(* LS Electric XG5000 project: Three_Guys_Plc *)
(* PLC LSPLC *)
(* module base 0 slot 0: FEnet:XGL-EFMT(B) (Fast Ethernet 통신 모듈, 전기 Master) *)
(* module base 0 slot 1: 입력 모듈:XGI-A21A/C (AC 220V 입력, 8점(8점/COM) / 8점(1점/COM)) *)
(* module base 0 slot 2: 출력 모듈:XGQ-RY1A (릴레이 출력, 8점 (2A용, 단독 COM.)) *)

PROGRAM HeatTreatPlc (* task: 스캔 프로그램 *)
VAR
    ENO : BOOL;
    곱하기60 : TIME := T#60s;
    기계1_가스_밸브 AT %MX8010 : BOOL;
    기계1_가스이상램프 AT %MX8011 : BOOL;
    기계1_가스이상센서 AT %MX8061 : BOOL;
    기계1_가열_min : TIME;
    기계1_가열_시간 AT %MD506 : DWORD;
    기계1_가열냉각_시간 : TIME;
    기계1_가열시간설정 : TOF;
    기계1_경고 AT %MX8019 : BOOL;
    기계1_경과시간_msec : TIME;
    기계1_남은시간_min AT %MD509 : TIME;
    기계1_남은시간_msec : TIME;
    기계1_냉각_min : TIME;
    기계1_냉각_밸브 AT %MX8012 : BOOL;
    기계1_냉각_시간 AT %MD507 : DWORD;
    기계1_냉각시간설정 : TOF;
    기계1_냉각이상램프 AT %MX8013 : BOOL;
    기계1_냉각이상센서 AT %MX8062 : BOOL;
    기계1_문 AT %MX8016 : BOOL;
    기계1_문ON_타이머 : TON;
    기계1_문이상램프 AT %MX8017 : BOOL;
    기계1_문이상센서 AT %MX8064 : BOOL;
    기계1_설정온도입력 AT %MW1010 : WORD;
    기계1_열선 AT %MX8014 : BOOL;
    기계1_열선이상램프 AT %MX8015 : BOOL;
    기계1_열선이상센서 AT %MX8063 : BOOL;
    기계1_작동 AT %MX8018 : BOOL;
    기계1_전원 AT %MX8001 : BOOL;
    기계1_중지 AT %MX8020 : BOOL;
    기계1_현재질화로온도 AT %MW1016 : WORD := 100;
    기계2_가스_밸브 AT %MX9010 : BOOL;
    기계2_가스이상램프 AT %MX9011 : BOOL;
    기계2_가스이상센서 AT %MX9061 : BOOL;
    기계2_가열_min : TIME;
    기계2_가열_시간 AT %MD569 : DWORD;
    기계2_가열냉각_시간 : TIME;
    기계2_가열시간설정 : TOF;
    기계2_경고 AT %MX9019 : BOOL;
    기계2_경과시간_msec : TIME;
    기계2_남은시간_min AT %MD572 : TIME;
    기계2_남은시간_msec : TIME;
    기계2_냉각_min : TIME;
    기계2_냉각_밸브 AT %MX9012 : BOOL;
    기계2_냉각_시간 AT %MD570 : DWORD;
    기계2_냉각시간설정 : TOF;
    기계2_냉각이상램프 AT %MX9013 : BOOL;
    기계2_냉각이상센서 AT %MX9062 : BOOL;
    기계2_문 AT %MX9016 : BOOL;
    기계2_문ON_타이머 : TON;
    기계2_문이상램프 AT %MX9017 : BOOL;
    기계2_문이상센서 AT %MX9064 : BOOL;
    기계2_설정온도입력 AT %MW1136 : WORD;
    기계2_열선 AT %MX9014 : BOOL;
    기계2_열선이상램프 AT %MX9015 : BOOL;
    기계2_열선이상센서 AT %MX9063 : BOOL;
    기계2_작동 AT %MX9018 : BOOL;
    기계2_전원 AT %MX9001 : BOOL;
    기계2_중지 AT %MX9020 : BOOL;
    기계2_현재질화로온도 AT %MW1142 : WORD;
    기계3_가스_밸브 AT %MX10010 : BOOL;
    기계3_가스이상램프 AT %MX10011 : BOOL;
    기계3_가스이상센서 AT %MX10061 : BOOL;
    기계3_가열_min : TIME;
    기계3_가열_시간 AT %MD631 : DWORD;
    기계3_가열냉각_시간 : TIME;
    기계3_가열시간설정 : TOF;
    기계3_경고 AT %MX10019 : BOOL;
    기계3_경과시간_msec : TIME;
    기계3_남은시간_min AT %MD634 : TIME;
    기계3_남은시간_msec : TIME;
    기계3_냉각_min : TIME;
    기계3_냉각_밸브 AT %MX10012 : BOOL;
    기계3_냉각_시간 AT %MD632 : DWORD;
    기계3_냉각시간설정 : TOF;
    기계3_냉각이상램프 AT %MX10013 : BOOL;
    기계3_냉각이상센서 AT %MX10062 : BOOL;
    기계3_문 AT %MX10016 : BOOL;
    기계3_문ON_타이머 : TON;
    기계3_문이상램프 AT %MX10017 : BOOL;
    기계3_문이상센서 AT %MX10064 : BOOL;
    기계3_설정온도입력 AT %MW1260 : WORD;
    기계3_열선 AT %MX10014 : BOOL;
    기계3_열선이상램프 AT %MX10015 : BOOL;
    기계3_열선이상센서 AT %MX10063 : BOOL;
    기계3_작동 AT %MX10018 : BOOL;
    기계3_전원 AT %MX10001 : BOOL;
    기계3_중지 AT %MX10020 : BOOL;
    기계3_현재질화로온도 AT %MW1266 : WORD;
    기계4_가스_밸브 AT %MX11010 : BOOL;
    기계4_가스이상램프 AT %MX11011 : BOOL;
    기계4_가스이상센서 AT %MX11061 : BOOL;
    기계4_가열_min : TIME;
    기계4_가열_시간 AT %MD694 : DWORD;
    기계4_가열냉각_시간 : TIME;
    기계4_가열시간설정 : TOF;
    기계4_경고 AT %MX11019 : BOOL;
    기계4_경과시간_msec : TIME;
    기계4_남은시간_min AT %MD697 : TIME;
    기계4_남은시간_msec : TIME;
    기계4_냉각_min : TIME;
    기계4_냉각_밸브 AT %MX11012 : BOOL;
    기계4_냉각_시간 AT %MD695 : DWORD;
    기계4_냉각시간설정 : TOF;
    기계4_냉각이상램프 AT %MX11013 : BOOL;
    기계4_냉각이상센서 AT %MX11062 : BOOL;
    기계4_문 AT %MX11016 : BOOL;
    기계4_문ON_타이머 : TON;
    기계4_문이상램프 AT %MX11017 : BOOL;
    기계4_문이상센서 AT %MX11064 : BOOL;
    기계4_설정온도입력 AT %MW1386 : WORD;
    기계4_열선 AT %MX11014 : BOOL;
    기계4_열선이상램프 AT %MX11015 : BOOL;
    기계4_열선이상센서 AT %MX11063 : BOOL;
    기계4_작동 AT %MX11018 : BOOL;
    기계4_전원 AT %MX11001 : BOOL;
    기계4_중지 AT %MX11020 : BOOL;
    기계4_현재질화로온도 AT %MW1392 : WORD;
    기계_신호기 : TP;
    기계_신호기1 : TP;
    기계_신호기2 : TP;
    기계_신호기3 : TP;
END_VAR
VAR
    _p1 : BOOL;
    _e2 : R_TRIG;
    _e3 : F_TRIG;
    _p4 : BOOL;
    _e5 : R_TRIG;
    _e6 : F_TRIG;
    _p7 : BOOL;
    _e8 : R_TRIG;
    _e9 : F_TRIG;
    _p10 : BOOL;
    _e11 : R_TRIG;
    _e12 : F_TRIG;
    _p13 : BOOL;
    _e14 : R_TRIG;
    _t15 : BOOL;
    _e16 : R_TRIG;
    _p17 : BOOL;
    _e18 : R_TRIG;
    _e19 : F_TRIG;
    _p20 : BOOL;
    _e21 : R_TRIG;
    _e22 : F_TRIG;
    _p23 : BOOL;
    _e24 : R_TRIG;
    _e25 : F_TRIG;
    _p26 : BOOL;
    _e27 : R_TRIG;
    _e28 : F_TRIG;
    _p29 : BOOL;
    _e30 : R_TRIG;
    _t31 : BOOL;
    _e32 : R_TRIG;
    _p33 : BOOL;
    _e34 : R_TRIG;
    _e35 : F_TRIG;
    _p36 : BOOL;
    _e37 : R_TRIG;
    _e38 : F_TRIG;
    _p39 : BOOL;
    _e40 : R_TRIG;
    _e41 : F_TRIG;
    _p42 : BOOL;
    _e43 : R_TRIG;
    _e44 : F_TRIG;
    _p45 : BOOL;
    _e46 : R_TRIG;
    _t47 : BOOL;
    _e48 : R_TRIG;
    _p49 : BOOL;
    _e50 : R_TRIG;
    _e51 : F_TRIG;
    _p52 : BOOL;
    _e53 : R_TRIG;
    _e54 : F_TRIG;
    _p55 : BOOL;
    _e56 : R_TRIG;
    _e57 : F_TRIG;
    _p58 : BOOL;
    _e59 : R_TRIG;
    _e60 : F_TRIG;
    _p61 : BOOL;
    _e62 : R_TRIG;
    _t63 : BOOL;
    _e64 : R_TRIG;
END_VAR

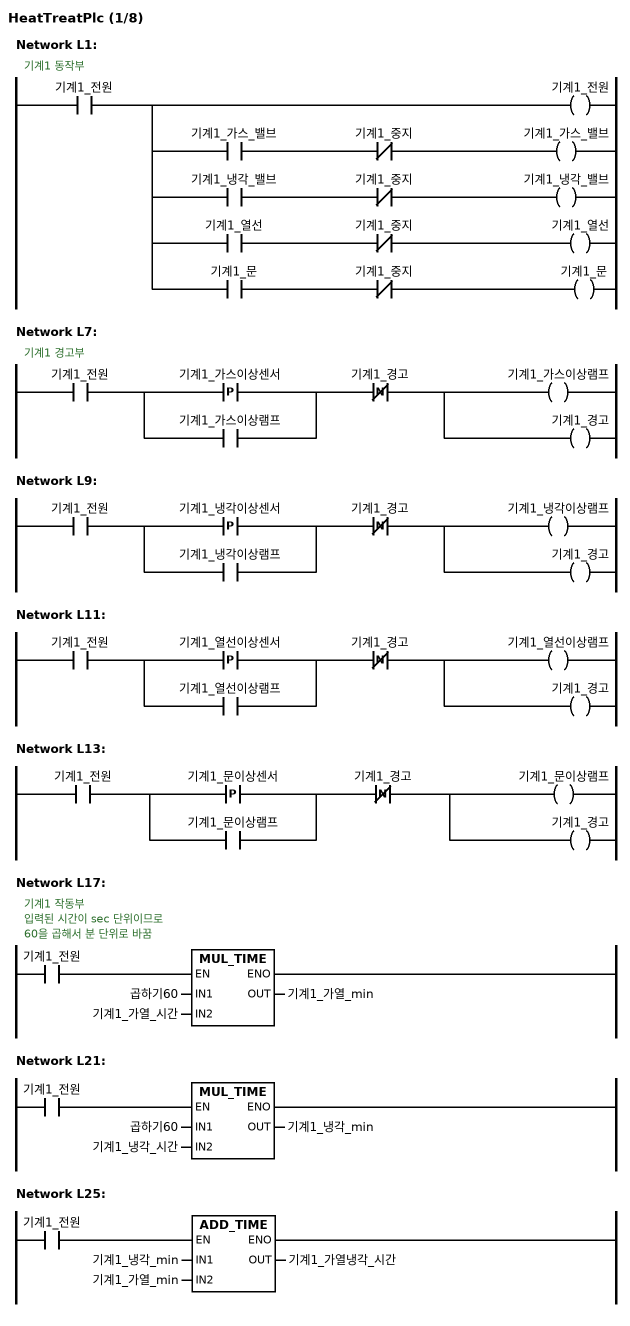
(* 기계1 동작부 *)
(* Rung L1 *)
_p1 := 기계1_전원;
기계1_전원 := _p1;
기계1_가스_밸브 := _p1 AND 기계1_가스_밸브 AND NOT 기계1_중지;
기계1_냉각_밸브 := _p1 AND 기계1_냉각_밸브 AND NOT 기계1_중지;
기계1_열선 := _p1 AND 기계1_열선 AND NOT 기계1_중지;
기계1_문 := _p1 AND 기계1_문 AND NOT 기계1_중지;
(* 기계1 경고부 *)
(* Rung L7 *)
_e2(CLK := 기계1_가스이상센서);
_e3(CLK := 기계1_경고);
_p4 := 기계1_전원 AND (_e2.Q OR 기계1_가스이상램프) AND NOT _e3.Q;
기계1_가스이상램프 := _p4;
기계1_경고 := _p4;
(* Rung L9 *)
_e5(CLK := 기계1_냉각이상센서);
_e6(CLK := 기계1_경고);
_p7 := 기계1_전원 AND (_e5.Q OR 기계1_냉각이상램프) AND NOT _e6.Q;
기계1_냉각이상램프 := _p7;
기계1_경고 := _p7;
(* Rung L11 *)
_e8(CLK := 기계1_열선이상센서);
_e9(CLK := 기계1_경고);
_p10 := 기계1_전원 AND (_e8.Q OR 기계1_열선이상램프) AND NOT _e9.Q;
기계1_열선이상램프 := _p10;
기계1_경고 := _p10;
(* Rung L13 *)
_e11(CLK := 기계1_문이상센서);
_e12(CLK := 기계1_경고);
_p13 := 기계1_전원 AND (_e11.Q OR 기계1_문이상램프) AND NOT _e12.Q;
기계1_문이상램프 := _p13;
기계1_경고 := _p13;
(* 기계1 작동부 *)
(* 입력된 시간이 sec 단위이므로 / 60을 곱해서 분 단위로 바꿈 *)
(* Rung L17 *)
IF 기계1_전원 THEN 기계1_가열_min := MUL_TIME(곱하기60, 기계1_가열_시간); END_IF;
(* Rung L21 *)
IF 기계1_전원 THEN 기계1_냉각_min := MUL_TIME(곱하기60, 기계1_냉각_시간); END_IF;
(* Rung L25 *)
IF 기계1_전원 THEN 기계1_가열냉각_시간 := ADD_TIME(기계1_냉각_min, 기계1_가열_min); END_IF;

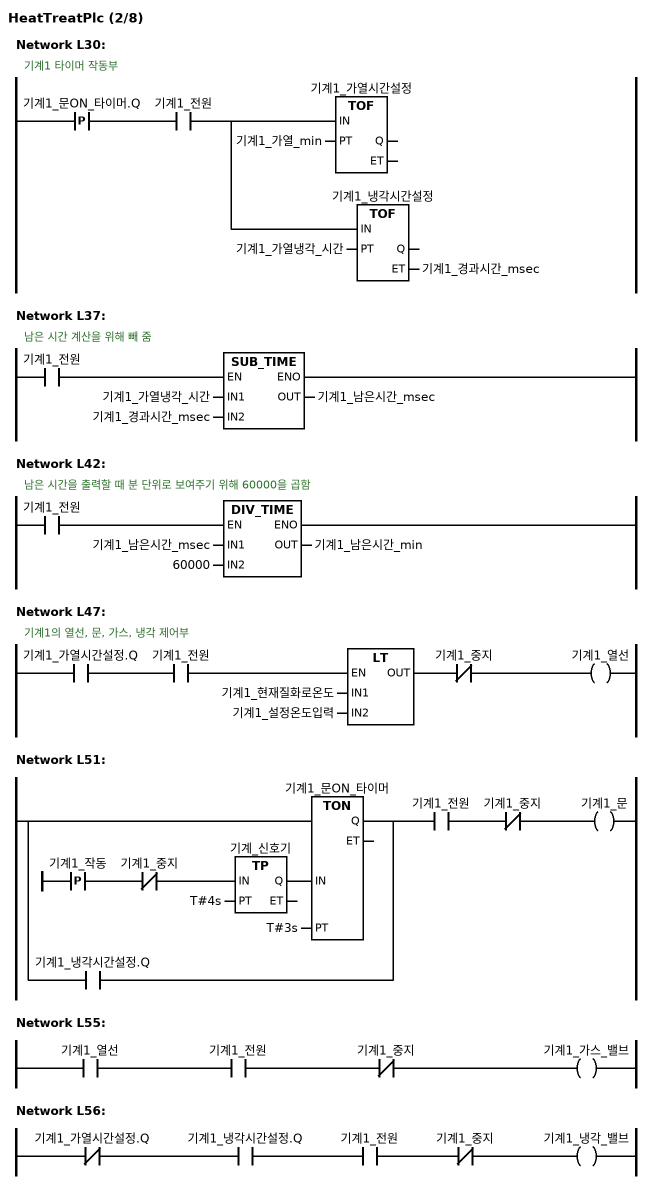
(* 기계1 타이머 작동부 *)
(* Rung L30 *)
_e14(CLK := 기계1_문ON_타이머.Q);
기계1_가열시간설정(IN := _e14.Q AND 기계1_전원, PT := 기계1_가열_min);
기계1_냉각시간설정(IN := _e14.Q AND 기계1_전원, PT := 기계1_가열냉각_시간, ET => 기계1_경과시간_msec);
(* 남은 시간 계산을 위해 빼 줌 *)
(* Rung L37 *)
IF 기계1_전원 THEN 기계1_남은시간_msec := SUB_TIME(기계1_가열냉각_시간, 기계1_경과시간_msec); END_IF;
(* 남은 시간을 출력할 때 분 단위로 보여주기 위해 60000을 곱함 *)
(* Rung L42 *)
IF 기계1_전원 THEN 기계1_남은시간_min := DIV_TIME(기계1_남은시간_msec, 60000); END_IF;
(* 기계1의 열선, 문, 가스, 냉각 제어부 *)
(* Rung L47 *)
IF 기계1_가열시간설정.Q AND 기계1_전원 THEN _t15 := 기계1_현재질화로온도 < 기계1_설정온도입력; END_IF;
기계1_열선 := _t15 AND NOT 기계1_중지;
(* Rung L51 *)
_e16(CLK := 기계1_작동);
기계_신호기(IN := _e16.Q AND NOT 기계1_중지, PT := T#4s);
기계1_문ON_타이머(IN := 기계_신호기.Q, PT := T#3s);
기계1_문 := (기계1_문ON_타이머.Q OR 기계1_냉각시간설정.Q) AND 기계1_전원 AND NOT 기계1_중지;
(* Rung L55 *)
기계1_가스_밸브 := 기계1_열선 AND 기계1_전원 AND NOT 기계1_중지;
(* Rung L56 *)
기계1_냉각_밸브 := NOT 기계1_가열시간설정.Q AND 기계1_냉각시간설정.Q AND 기계1_전원 AND NOT 기계1_중지;

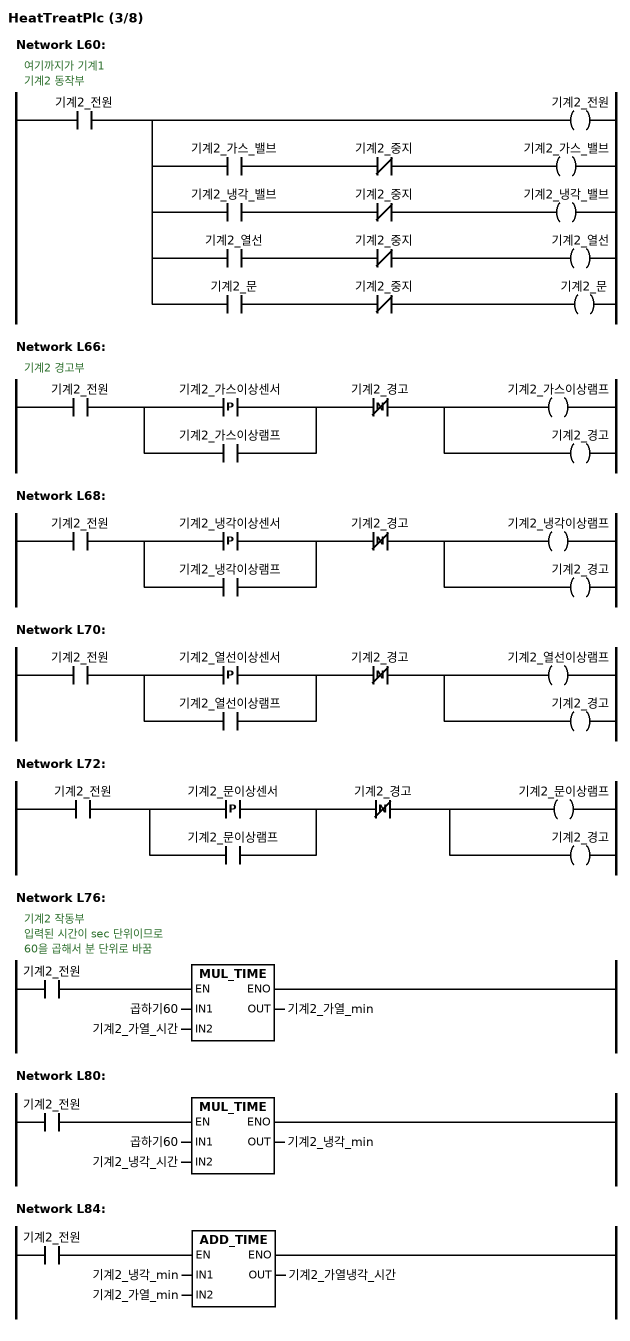
(* 여기까지가 기계1 *)
(* 기계2 동작부 *)
(* Rung L60 *)
_p17 := 기계2_전원;
기계2_전원 := _p17;
기계2_가스_밸브 := _p17 AND 기계2_가스_밸브 AND NOT 기계2_중지;
기계2_냉각_밸브 := _p17 AND 기계2_냉각_밸브 AND NOT 기계2_중지;
기계2_열선 := _p17 AND 기계2_열선 AND NOT 기계2_중지;
기계2_문 := _p17 AND 기계2_문 AND NOT 기계2_중지;
(* 기계2 경고부 *)
(* Rung L66 *)
_e18(CLK := 기계2_가스이상센서);
_e19(CLK := 기계2_경고);
_p20 := 기계2_전원 AND (_e18.Q OR 기계2_가스이상램프) AND NOT _e19.Q;
기계2_가스이상램프 := _p20;
기계2_경고 := _p20;
(* Rung L68 *)
_e21(CLK := 기계2_냉각이상센서);
_e22(CLK := 기계2_경고);
_p23 := 기계2_전원 AND (_e21.Q OR 기계2_냉각이상램프) AND NOT _e22.Q;
기계2_냉각이상램프 := _p23;
기계2_경고 := _p23;
(* Rung L70 *)
_e24(CLK := 기계2_열선이상센서);
_e25(CLK := 기계2_경고);
_p26 := 기계2_전원 AND (_e24.Q OR 기계2_열선이상램프) AND NOT _e25.Q;
기계2_열선이상램프 := _p26;
기계2_경고 := _p26;
(* Rung L72 *)
_e27(CLK := 기계2_문이상센서);
_e28(CLK := 기계2_경고);
_p29 := 기계2_전원 AND (_e27.Q OR 기계2_문이상램프) AND NOT _e28.Q;
기계2_문이상램프 := _p29;
기계2_경고 := _p29;
(* 기계2 작동부 *)
(* 입력된 시간이 sec 단위이므로 / 60을 곱해서 분 단위로 바꿈 *)
(* Rung L76 *)
IF 기계2_전원 THEN 기계2_가열_min := MUL_TIME(곱하기60, 기계2_가열_시간); END_IF;
(* Rung L80 *)
IF 기계2_전원 THEN 기계2_냉각_min := MUL_TIME(곱하기60, 기계2_냉각_시간); END_IF;
(* Rung L84 *)
IF 기계2_전원 THEN 기계2_가열냉각_시간 := ADD_TIME(기계2_냉각_min, 기계2_가열_min); END_IF;

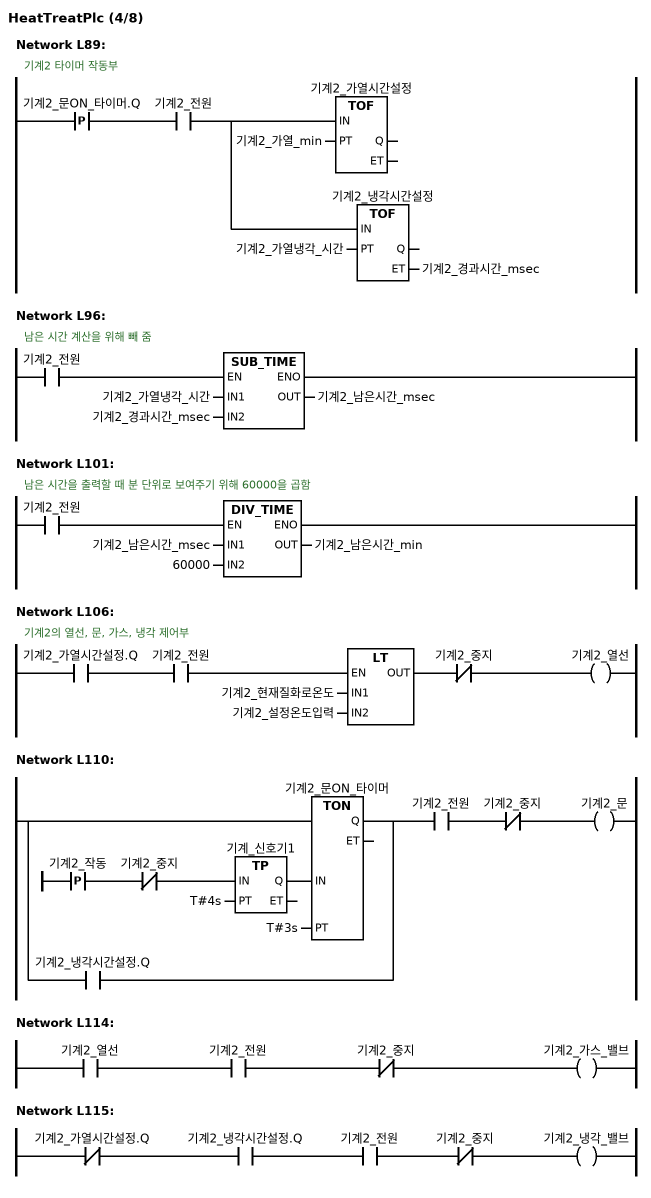
(* 기계2 타이머 작동부 *)
(* Rung L89 *)
_e30(CLK := 기계2_문ON_타이머.Q);
기계2_가열시간설정(IN := _e30.Q AND 기계2_전원, PT := 기계2_가열_min);
기계2_냉각시간설정(IN := _e30.Q AND 기계2_전원, PT := 기계2_가열냉각_시간, ET => 기계2_경과시간_msec);
(* 남은 시간 계산을 위해 빼 줌 *)
(* Rung L96 *)
IF 기계2_전원 THEN 기계2_남은시간_msec := SUB_TIME(기계2_가열냉각_시간, 기계2_경과시간_msec); END_IF;
(* 남은 시간을 출력할 때 분 단위로 보여주기 위해 60000을 곱함 *)
(* Rung L101 *)
IF 기계2_전원 THEN 기계2_남은시간_min := DIV_TIME(기계2_남은시간_msec, 60000); END_IF;
(* 기계2의 열선, 문, 가스, 냉각 제어부 *)
(* Rung L106 *)
IF 기계2_가열시간설정.Q AND 기계2_전원 THEN _t31 := 기계2_현재질화로온도 < 기계2_설정온도입력; END_IF;
기계2_열선 := _t31 AND NOT 기계2_중지;
(* Rung L110 *)
_e32(CLK := 기계2_작동);
기계_신호기1(IN := _e32.Q AND NOT 기계2_중지, PT := T#4s);
기계2_문ON_타이머(IN := 기계_신호기1.Q, PT := T#3s);
기계2_문 := (기계2_문ON_타이머.Q OR 기계2_냉각시간설정.Q) AND 기계2_전원 AND NOT 기계2_중지;
(* Rung L114 *)
기계2_가스_밸브 := 기계2_열선 AND 기계2_전원 AND NOT 기계2_중지;
(* Rung L115 *)
기계2_냉각_밸브 := NOT 기계2_가열시간설정.Q AND 기계2_냉각시간설정.Q AND 기계2_전원 AND NOT 기계2_중지;

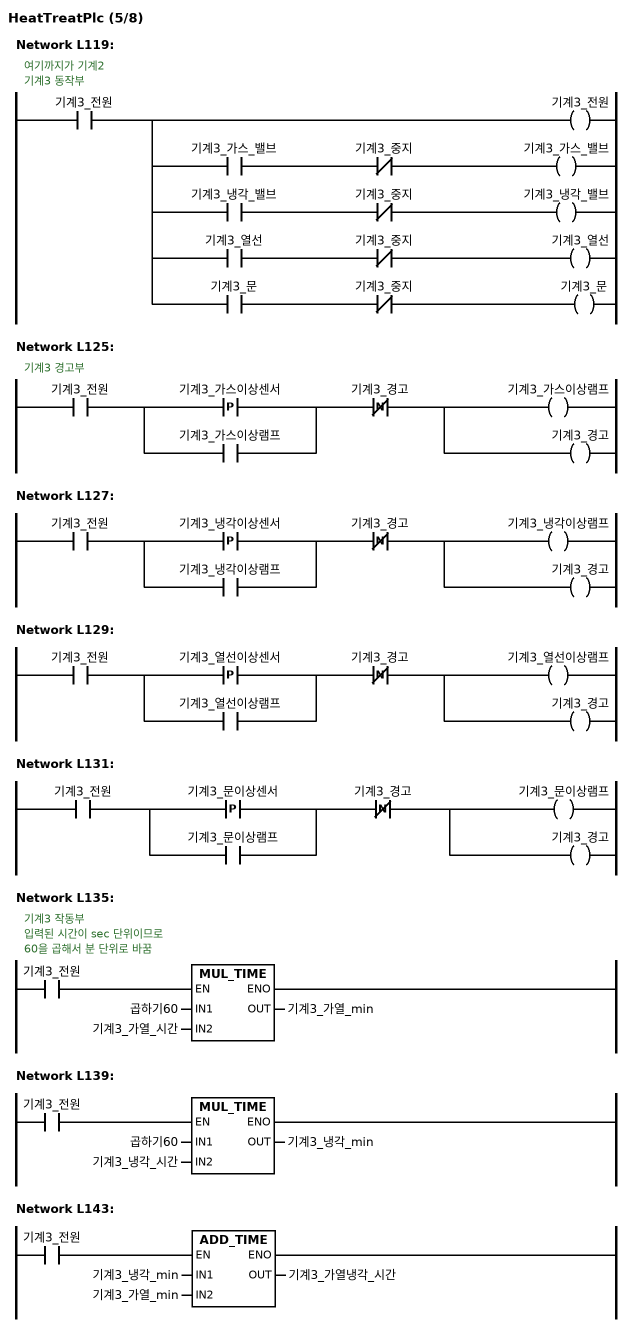
(* 여기까지가 기계2 *)
(* 기계3 동작부 *)
(* Rung L119 *)
_p33 := 기계3_전원;
기계3_전원 := _p33;
기계3_가스_밸브 := _p33 AND 기계3_가스_밸브 AND NOT 기계3_중지;
기계3_냉각_밸브 := _p33 AND 기계3_냉각_밸브 AND NOT 기계3_중지;
기계3_열선 := _p33 AND 기계3_열선 AND NOT 기계3_중지;
기계3_문 := _p33 AND 기계3_문 AND NOT 기계3_중지;
(* 기계3 경고부 *)
(* Rung L125 *)
_e34(CLK := 기계3_가스이상센서);
_e35(CLK := 기계3_경고);
_p36 := 기계3_전원 AND (_e34.Q OR 기계3_가스이상램프) AND NOT _e35.Q;
기계3_가스이상램프 := _p36;
기계3_경고 := _p36;
(* Rung L127 *)
_e37(CLK := 기계3_냉각이상센서);
_e38(CLK := 기계3_경고);
_p39 := 기계3_전원 AND (_e37.Q OR 기계3_냉각이상램프) AND NOT _e38.Q;
기계3_냉각이상램프 := _p39;
기계3_경고 := _p39;
(* Rung L129 *)
_e40(CLK := 기계3_열선이상센서);
_e41(CLK := 기계3_경고);
_p42 := 기계3_전원 AND (_e40.Q OR 기계3_열선이상램프) AND NOT _e41.Q;
기계3_열선이상램프 := _p42;
기계3_경고 := _p42;
(* Rung L131 *)
_e43(CLK := 기계3_문이상센서);
_e44(CLK := 기계3_경고);
_p45 := 기계3_전원 AND (_e43.Q OR 기계3_문이상램프) AND NOT _e44.Q;
기계3_문이상램프 := _p45;
기계3_경고 := _p45;
(* 기계3 작동부 *)
(* 입력된 시간이 sec 단위이므로 / 60을 곱해서 분 단위로 바꿈 *)
(* Rung L135 *)
IF 기계3_전원 THEN 기계3_가열_min := MUL_TIME(곱하기60, 기계3_가열_시간); END_IF;
(* Rung L139 *)
IF 기계3_전원 THEN 기계3_냉각_min := MUL_TIME(곱하기60, 기계3_냉각_시간); END_IF;
(* Rung L143 *)
IF 기계3_전원 THEN 기계3_가열냉각_시간 := ADD_TIME(기계3_냉각_min, 기계3_가열_min); END_IF;

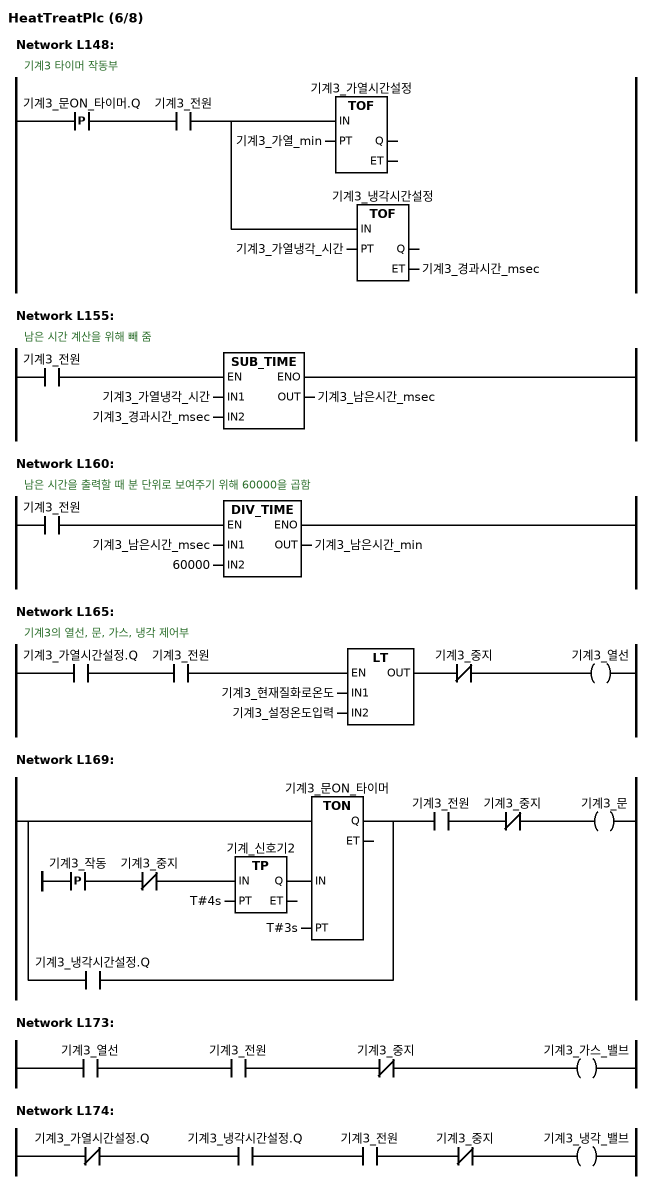
(* 기계3 타이머 작동부 *)
(* Rung L148 *)
_e46(CLK := 기계3_문ON_타이머.Q);
기계3_가열시간설정(IN := _e46.Q AND 기계3_전원, PT := 기계3_가열_min);
기계3_냉각시간설정(IN := _e46.Q AND 기계3_전원, PT := 기계3_가열냉각_시간, ET => 기계3_경과시간_msec);
(* 남은 시간 계산을 위해 빼 줌 *)
(* Rung L155 *)
IF 기계3_전원 THEN 기계3_남은시간_msec := SUB_TIME(기계3_가열냉각_시간, 기계3_경과시간_msec); END_IF;
(* 남은 시간을 출력할 때 분 단위로 보여주기 위해 60000을 곱함 *)
(* Rung L160 *)
IF 기계3_전원 THEN 기계3_남은시간_min := DIV_TIME(기계3_남은시간_msec, 60000); END_IF;
(* 기계3의 열선, 문, 가스, 냉각 제어부 *)
(* Rung L165 *)
IF 기계3_가열시간설정.Q AND 기계3_전원 THEN _t47 := 기계3_현재질화로온도 < 기계3_설정온도입력; END_IF;
기계3_열선 := _t47 AND NOT 기계3_중지;
(* Rung L169 *)
_e48(CLK := 기계3_작동);
기계_신호기2(IN := _e48.Q AND NOT 기계3_중지, PT := T#4s);
기계3_문ON_타이머(IN := 기계_신호기2.Q, PT := T#3s);
기계3_문 := (기계3_문ON_타이머.Q OR 기계3_냉각시간설정.Q) AND 기계3_전원 AND NOT 기계3_중지;
(* Rung L173 *)
기계3_가스_밸브 := 기계3_열선 AND 기계3_전원 AND NOT 기계3_중지;
(* Rung L174 *)
기계3_냉각_밸브 := NOT 기계3_가열시간설정.Q AND 기계3_냉각시간설정.Q AND 기계3_전원 AND NOT 기계3_중지;

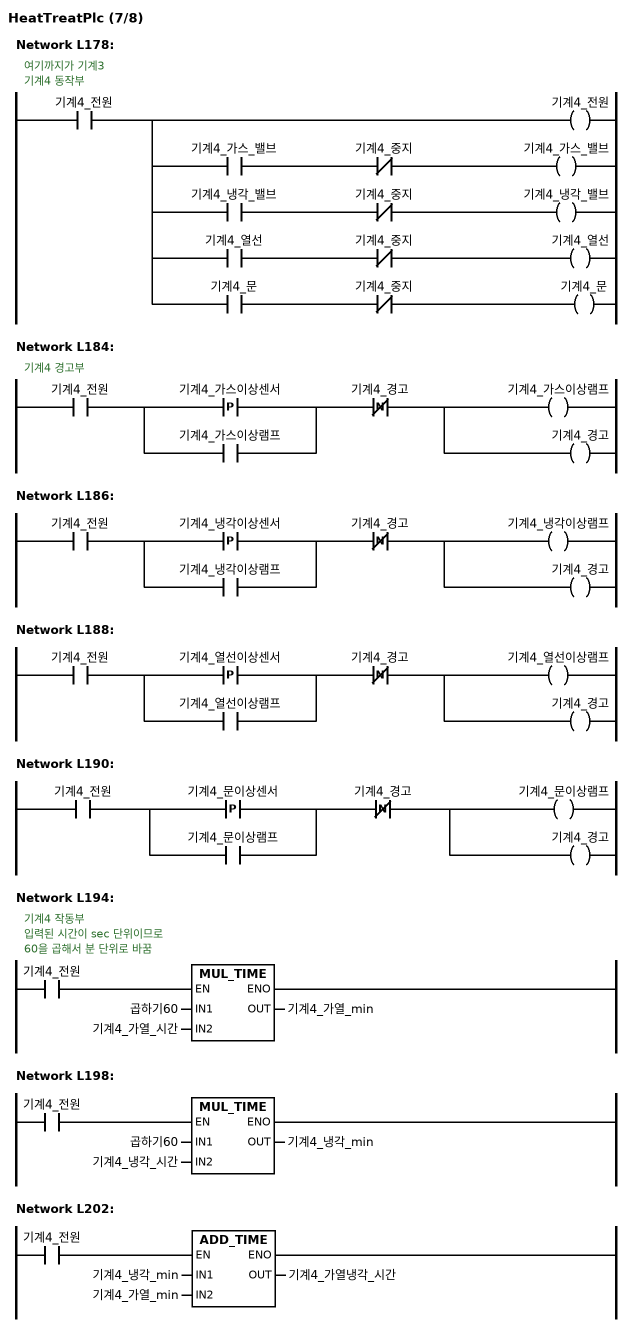
(* 여기까지가 기계3 *)
(* 기계4 동작부 *)
(* Rung L178 *)
_p49 := 기계4_전원;
기계4_전원 := _p49;
기계4_가스_밸브 := _p49 AND 기계4_가스_밸브 AND NOT 기계4_중지;
기계4_냉각_밸브 := _p49 AND 기계4_냉각_밸브 AND NOT 기계4_중지;
기계4_열선 := _p49 AND 기계4_열선 AND NOT 기계4_중지;
기계4_문 := _p49 AND 기계4_문 AND NOT 기계4_중지;
(* 기계4 경고부 *)
(* Rung L184 *)
_e50(CLK := 기계4_가스이상센서);
_e51(CLK := 기계4_경고);
_p52 := 기계4_전원 AND (_e50.Q OR 기계4_가스이상램프) AND NOT _e51.Q;
기계4_가스이상램프 := _p52;
기계4_경고 := _p52;
(* Rung L186 *)
_e53(CLK := 기계4_냉각이상센서);
_e54(CLK := 기계4_경고);
_p55 := 기계4_전원 AND (_e53.Q OR 기계4_냉각이상램프) AND NOT _e54.Q;
기계4_냉각이상램프 := _p55;
기계4_경고 := _p55;
(* Rung L188 *)
_e56(CLK := 기계4_열선이상센서);
_e57(CLK := 기계4_경고);
_p58 := 기계4_전원 AND (_e56.Q OR 기계4_열선이상램프) AND NOT _e57.Q;
기계4_열선이상램프 := _p58;
기계4_경고 := _p58;
(* Rung L190 *)
_e59(CLK := 기계4_문이상센서);
_e60(CLK := 기계4_경고);
_p61 := 기계4_전원 AND (_e59.Q OR 기계4_문이상램프) AND NOT _e60.Q;
기계4_문이상램프 := _p61;
기계4_경고 := _p61;
(* 기계4 작동부 *)
(* 입력된 시간이 sec 단위이므로 / 60을 곱해서 분 단위로 바꿈 *)
(* Rung L194 *)
IF 기계4_전원 THEN 기계4_가열_min := MUL_TIME(곱하기60, 기계4_가열_시간); END_IF;
(* Rung L198 *)
IF 기계4_전원 THEN 기계4_냉각_min := MUL_TIME(곱하기60, 기계4_냉각_시간); END_IF;
(* Rung L202 *)
IF 기계4_전원 THEN 기계4_가열냉각_시간 := ADD_TIME(기계4_냉각_min, 기계4_가열_min); END_IF;

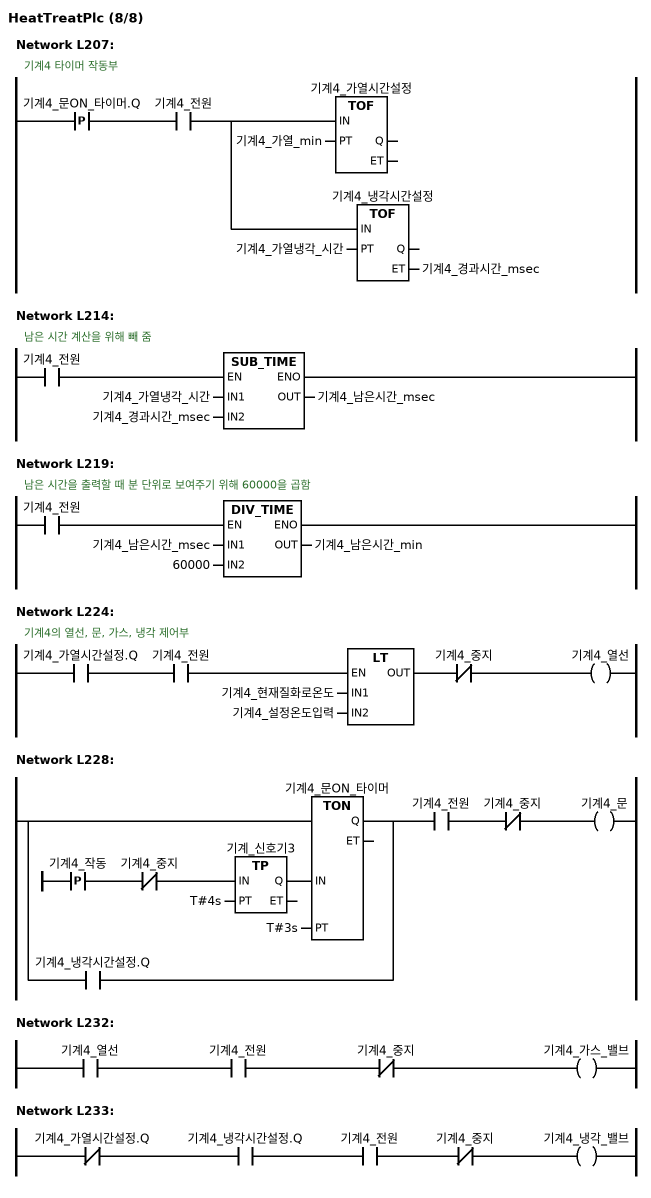
(* 기계4 타이머 작동부 *)
(* Rung L207 *)
_e62(CLK := 기계4_문ON_타이머.Q);
기계4_가열시간설정(IN := _e62.Q AND 기계4_전원, PT := 기계4_가열_min);
기계4_냉각시간설정(IN := _e62.Q AND 기계4_전원, PT := 기계4_가열냉각_시간, ET => 기계4_경과시간_msec);
(* 남은 시간 계산을 위해 빼 줌 *)
(* Rung L214 *)
IF 기계4_전원 THEN 기계4_남은시간_msec := SUB_TIME(기계4_가열냉각_시간, 기계4_경과시간_msec); END_IF;
(* 남은 시간을 출력할 때 분 단위로 보여주기 위해 60000을 곱함 *)
(* Rung L219 *)
IF 기계4_전원 THEN 기계4_남은시간_min := DIV_TIME(기계4_남은시간_msec, 60000); END_IF;
(* 기계4의 열선, 문, 가스, 냉각 제어부 *)
(* Rung L224 *)
IF 기계4_가열시간설정.Q AND 기계4_전원 THEN _t63 := 기계4_현재질화로온도 < 기계4_설정온도입력; END_IF;
기계4_열선 := _t63 AND NOT 기계4_중지;
(* Rung L228 *)
_e64(CLK := 기계4_작동);
기계_신호기3(IN := _e64.Q AND NOT 기계4_중지, PT := T#4s);
기계4_문ON_타이머(IN := 기계_신호기3.Q, PT := T#3s);
기계4_문 := (기계4_문ON_타이머.Q OR 기계4_냉각시간설정.Q) AND 기계4_전원 AND NOT 기계4_중지;
(* Rung L232 *)
기계4_가스_밸브 := 기계4_열선 AND 기계4_전원 AND NOT 기계4_중지;
(* Rung L233 *)
기계4_냉각_밸브 := NOT 기계4_가열시간설정.Q AND 기계4_냉각시간설정.Q AND 기계4_전원 AND NOT 기계4_중지;
END_PROGRAM